# EPICS autosave request: ADPointGrey/pointGreyApp/Db/pointGreyProperty_settings.req
$(P)$(R)$(PROPERTY)OnOff
$(P)$(R)$(PROPERTY)Val
$(P)$(R)$(PROPERTY)ValB
$(P)$(R)$(PROPERTY)ValAbs
$(P)$(R)$(PROPERTY)AutoMode
